// TIA Portal V20 export
DATA_BLOCK "SBK01"   // DB322
// stored: MemoryReserve 100
   VAR
      "EMO01 CH.A" : Bool;
      "EMO02 CH.A" : Bool;
      SPARE : Bool;
      "EMO04 CH.A" : Bool;
      "EMO01 CH.B" : Bool;
      "EMO02 CH.B" : Bool;
      SPARE_1 : Bool;
      "EMO04 CH.B" : Bool;
      SPARE_2 : Bool;
      SPARE_3 : Bool;
      SPARE_4 : Bool;
   END_VAR
BEGIN
END_DATA_BLOCK
